PROGRAM MAIN
VAR
END_VAR

END_PROGRAM

(* stored: Version 1.1.0.1
   POU MAIN: Id {2fa6ab45-28f7-4a9f-8627-4602397d4832} *)
